Staubli VAL3: Cognex.pjx

--- Cognex.pjx ---
Parameters version=s7.4 stackSize=5000 millimeterUnit=true
Program file=checkCellFormat.pgx
Program file=checkColValue.pgx
Program file=checkErrFormat.pgx
Program file=debugMsg.pgx
Program file=example.pgx
Program file=getErrorCode.pgx
Program file=getErrorMessage.pgx
Program file=getFile.pgx
Program file=getFullError.pgx
Program file=getLibVersion.pgx
Program file=getNextID.pgx
Program file=getOnline.pgx
Program file=incrementCol.pgx
Program file=init.pgx
Program file=initPUPITRE.pgx
Program file=isIDAvailable.pgx
Program file=isLoggedIn.pgx
Program file=loadFile.pgx
Program file=login.pgx
Program file=programmeMOVE.pgx
Program file=readLogin.pgx
Program file=readNumValue.pgx
Program file=readRect.pgx
Program file=readSocket.pgx
Program file=readStrValue.pgx
Program file=readTrsf.pgx
Program file=readme.pgx
Program file=safety.pgx
Program file=saveFile.pgx
Program file=sendCommand.pgx
Program file=setCheckRow.pgx
Program file=setEventAndWait.pgx
Program file=setEventNoWait.pgx
Program file=setIDAutoMgt.pgx
Program file=setOnline.pgx
Program file=start.pgx
Program file=stop.pgx
Program file=trigger.pgx
Program file=writeFloatValue.pgx
Program file=writeIntValue.pgx
Program file=writeSocket.pgx
Program file=writeStrValue.pgx
Data file=Cognex.dtx
Type name=camera path=./camera/camera.pjx

--- checkCellFormat.pgx ---
public program checkCellFormat(num x_nCamID (dimensions=1), string& x_sCellNumber[] (dimensions=1), bool& x_bMatchOk[] (dimensions=1))
  local num l_i
  local bool l_bColOk
  local bool l_bRowOk
  local string l_sColumn
  local string l_sRow
  local num l_nRow
  local num l_nError
  local string l_sMsgError
begin
  //-----------------------------------------------------------------------
  //Header begin
  //Description of program
  // This routines checks if the format of the string used to point on a cell
  // of the cognex speadsheet matches the format of native command.
  //
  // Input Parameters
  //  x_nCamID :
  //    role : camera's ID
  //   x_sCellNumber  :
  //     role : Cell number in string format.
  //            Must be : - First digit is a letter (A-Z) for Column number
  //                      - 3 next digits is a number for Row number
  //
  // Output Parameteres
  //  x_bMatchOK  :
  //    role : retruns true if format of the string x_sCellNumber is correct
  //          and false otherwise.
  //
  //Examples
  //  call checkCellFormat(nCamID,"A3",l_bCellOk)
  //
  //Header end
  //-----------------------------------------------------------------------

  //Init
  x_bMatchOk=false
  //Verify length of the string (minimum 2 digit, ex : "A1")
  if len(x_sCellNumber)>=2
    //Column of the CellNumber
    l_sColumn=left(x_sCellNumber,1)
    //Verify first digit (column)
    //First digit must be in range 'A-Z' or 'a-z'
    call checkColValue(l_sColumn,l_bColOk)
    if l_bColOk
      //First digit OK
      //Row of the CellNumber
      l_sRow=right(x_sCellNumber,len(x_sCellNumber)-1)
      toNum(l_sRow,l_nRow,l_bRowOk)
      if l_bRowOk
        //l_sRow is a numercial value
        //Verify the row number
        if l_nRow>=0 and (l_nRow<=400 or !bCheckRowUpLim)
          if len(l_sRow)<3
            //Add digits (there is always 3 digits)
            l_sRow=left("000",3-len(l_sRow))+l_sRow
            //Update CellNumber
            x_sCellNumber=l_sColumn+l_sRow
          endIf
          //Cell Format OK
          x_bMatchOk=true
          cCamera[x_nCamID].nErrorCode=110
        else
          //Row number out of range
          cCamera[x_nCamID].nErrorCode=113
          cCamera[x_nCamID].sErrorMsg[cCamera[x_nCamID].nErrorCode]="Cell Format> "+l_sRow+" row number out of range"
        endIf
      else
        //Invalid row (not a numerical value)
        cCamera[x_nCamID].nErrorCode=112
        cCamera[x_nCamID].sErrorMsg[cCamera[x_nCamID].nErrorCode]="Cell Format> "+l_sRow+" invalid row"
      endIf
    else
      //Invalid column
      cCamera[x_nCamID].nErrorCode=111
      cCamera[x_nCamID].sErrorMsg[cCamera[x_nCamID].nErrorCode]="Cell Format> "+l_sColumn+" invalid column"
    endIf
  endIf
  if bDebugProgram
    //Displays error message
    call getFullError(x_nCamID,l_nError,l_sMsgError)
    ? l_sMsgError
  endIf
end

--- checkColValue.pgx ---
public program checkColValue(string x_sColCharac (dimensions=1), bool& x_bColOk[] (dimensions=1))
begin
  //-----------------------------------------------------------------------
  //Header begin
  //Description of program
  //  Check the column number of the x_sCellNumber.
  //
  // Input Parameters
  //   x_sCellNumber  :
  //     role : cell number in string format.
  //            Must be : - First digit is a letter (A-Z) for Column number
  //                      - 3 next digits is a number for Row number
  //
  // Output Parameteres
  //  x_bColOk  :
  //    role : returns true if the operation succeeded and false
  //          otherwise
  //
  //Header end
  //-----------------------------------------------------------------------

  //Verify column character (between "A" to "Z" or "a" to "z")
  x_bColOk=(asc(x_sColCharac,0)>=asc("a",0)) and (asc(x_sColCharac,0)<=asc("z",0))
  x_bColOk=x_bColOk or (asc(x_sColCharac,0)>=asc("A",0)) and (asc(x_sColCharac,0)<=asc("Z",0))
end

--- getErrorCode.pgx ---
public program getErrorCode(num x_nCamID (dimensions=1), num& x_nErrorCode[] (dimensions=1))
begin
  //-----------------------------------------------------------------------
  //Header begin
  //Description of program
  //  Get error code of last executed command.
  //
  //Input parameters
  //  num x_nCamID :
  //    role : camera's ID
  //
  //Output parameters
  //  num x_nErrorCode :
  //    role : error code of the last executed command
  //
  //Examples
  //  call getErrorCode(nCamID,l_nErrorCode)
  //
  //History
  //  Creation : 19-05-08 - f.Rob
  //  Modification 06-2012 - T.Caille - C.Rocchini
  //Header end
  //-----------------------------------------------------------------------
  if nLibErrorCode==0
    x_nErrorCode=cCamera[x_nCamID].nErrorCode
  else
    x_nErrorCode=nLibErrorCode
    nLibErrorCode=0
  endIf
  nCamID=x_nCamID
end

--- getLibVersion.pgx ---
public program getLibVersion(string& x_sVersion[] (dimensions=1))
begin
  //-----------------------------------------------------------------------
  //Header begin
  //Description of program
  //  Retrieve version of the library.
  //
  //Output parameters
  //  string x_sVersion :
  //    role : version of the library
  //
  //Examples
  //  call getLibVersion(l_sLibVersion)
  //
  //History
  //  Creation : 19-05-08 - f.Rob
  //Header end
  //-----------------------------------------------------------------------

  x_sVersion=strVersion
end

--- incrementCol.pgx ---
public program incrementCol(string& x_sCellNumber[] (dimensions=1), bool& x_bColumnOK[] (dimensions=1))
  local string l_sColCharac
begin
  //-----------------------------------------------------------------------
  //Header begin
  //Description of program
  //  Increment the column number of the x_sCellNumber.
  //
  // Input Parameters
  //   x_sCellNumber  :
  //     role : Cell number in string format.
  //            Must be : - First digit is a letter (A-Z) for Column number
  //                      - 3 next digits is a number for Row number
  //
  // Output Parameteres
  //  x_bColumnOK  :
  //    role : returns true if the increment column is succeeded and false
  //          otherwise
  //
  //History
  //  Creation : 19-05-08 - f.Rob
  //  Modification : 10-07-08 - CROC
  //    correction of bug in the line that rebuilds the new incremented cell
  //    number, the line "right(x_sCellNumber,3)" has been replaced by
  //    "right(x_sCellNumber,len(x_sCellNumber)-1)" to be more flexible in
  //    regards to cell number format (before that the cell number had to be
  //    composed of one letter and 3 numbers, now the only restriction is that
  //    the first character has to be a letter). This modification was triggered
  //    by the fact that this procedure is used by readRect() that passes the
  //    cell numbers as 2 char only (one letter, one number), thus it wasn't
  //    working properly.
  //Header end
  //-----------------------------------------------------------------------

  //Get the number column
  l_sColCharac=left(x_sCellNumber,1)
  //Increment the number column
  l_sColCharac=chr((asc(l_sColCharac,0)+1))
  //Checks the number column ( A<Column<Z)
  call checkColValue(l_sColCharac,x_bColumnOK)
  if x_bColumnOK
    //Modify x_sCellNumber
    x_sCellNumber=l_sColCharac+right(x_sCellNumber,len(x_sCellNumber)-1)
  endIf
end

--- loadFile.pgx ---
public program loadFile(num x_nCamID (dimensions=1), string x_sNameJob (dimensions=1), bool& x_bError[] (dimensions=1))
begin
  //-----------------------------------------------------------------------
  //Header begin
  //Description of program
  //  Loads the specified job from flash memory on the In-Sight sensor,
  //  making it the active job.
  //
  //!!! The In-Sight sensor must be OFFLINE !!!
  //
  //Input parameters
  //  num x_nCamID :
  //    role : camera's ID
  //
  //Output parameters
  //  string x_sNameJob :
  //    role : The name of the job.
  //           The command will execute with or without the .JOB extension.
  //
  //  bool x_bError :
  //    role : returns true if an error occurred and false otherwise
  //
  //Examples
  //   call loadFile(nCamID,"Camera1.job",x_bError)
  //
  //History
  //  Creation : 19-05-08 - f.Rob
  //Header end
  //-----------------------------------------------------------------------

  nProgram[x_nCamID]=4
  call sendCommand(x_nCamID,"LF"+x_sNameJob,x_bError)
end

--- login.pgx ---
public program login(sio& x_sioSocket (dimensions=1), string x_sUser (dimensions=1), string x_sPassword (dimensions=1), num& x_nCamID (dimensions=1), bool& x_bError[] (dimensions=1))
  local string l_sMsg
  local bool l_bError
begin
  //-----------------------------------------------------------------------
  //Header begin
  //Description of program
  //  Login to camera via TCP/IP socket port 1023, password pair
  // (usually "admin" and "").
  //  Returns camera's ID of type num for further communication with the camera.
  //
  //Input parameters
  //  string x_sUser :
  //    role : user name
  //  string x_sPassword :
  //    role : password for the user x_sUser
  //
  //Output parameters
  //  sio x_sioSocket :
  //    role : CS8 client socket
  //  num x_nCamID :
  //    role : returns camera's ID for further operations as the lib can
  //          communicate with more that 1 camera.
  //    posssible values : - first camera (first login)  : x_nCamID=1
  //                       - second camera (second login): x_nCamID=2
  //                       - ...
  //  bool x_bError :
  //    role : returns true if an error occurred and false otherwise
  //
  //Examples
  //  call login(cognex1,"admin","",nCamID,x_bError)
  //
  //History
  //  Creation : 19-05-08 - f.Rob
  //Header end
  //-----------------------------------------------------------------------
  if bDebugProgram
    putln("Cognex login")
  endIf
  // Check available ID
  l_bError=false
  if bGetID==true
    call isIDAvailable(x_nCamID,l_bError)
  endIf
  if l_bError==false
    nProgram[x_nCamID]=1
    sioLink(cCamera[x_nCamID].sSocket,x_sioSocket)
    // Read welcome string
    call readSocket(x_nCamID,l_sMsg,x_bError)
    // Send user name
    call readLogin(x_nCamID,l_sMsg,x_bError)
    call writeSocket(x_nCamID,x_sUser)
    // Send password
    call readLogin(x_nCamID,l_sMsg,x_bError)
    call writeSocket(x_nCamID,x_sPassword)
    // Read login result
    call readSocket(x_nCamID,l_sMsg,x_bError)
    x_bError=find(l_sMsg,"User Logged In")==-1
    if x_bError
      cCamera[x_nCamID].nErrorCode=1
      cCamera[x_nCamID].bConnected=false
      if bDebugProgram
        putln("Login : failed")
      endIf
    else
      cCamera[x_nCamID].bConnected=true
    endIf
  else
    x_bError=true
    nLibErrorCode=203
  endIf
end

--- programmeMOVE.pgx ---
program programmeMOVE()
begin
  while true

    // boucle infini

    while (borange==true)
      // BOUCLE DE DEBOXAGE

      // DEMANDE UNE MISE EN LIGNE DE LA CAMERA SI CELLE SI EST ETEINTE
      call getOnline(nCamID,resultTrigger)
      //APPEL UNE CAPURE DE PHOTO
      call trigger(nCamID,l_bError)

      delay(1.5)



      // RECUPERATION DONNE DANS LE TABLEUR COGNEX DANS LES CELLULE CC36/D36/E36
      call readNumValue(nCamID,"C36",resultx,l_bError)
      call readNumValue(nCamID,"D36",resulty,l_bError)
      call readNumValue(nCamID,"E36",resultz,l_bError)


      nbPoint=nbPoint+1
      putln("COORDONNEE DU POINT :")
      putln(nbPoint)
      putln("Coordonnée X:")
      putln(resultx)
      putln("Coordonnée Y:")
      putln(resulty)
      putln("Coordonnée Z:")
      putln(resultz)


      // AFFECTATION DES VALEUR DE X Y Z DU POINT CAMERA QUI EST DANS LE FRAME CAMERA
      PointCamera.trsf.x=resultx
      PointCamera.trsf.y=resulty
      PointCamera.trsf.z=55.5
      PointCamera.trsf.rx=180
      PointCamera.trsf.ry=0
      PointCamera.trsf.rz=90



      close(pince)



      movej(appro(PointCamera,{0,0,-100,0,0,0}),pince,rapide)
      movel(PointCamera,pince,lent)




      delay(1)

      open(pince)

      delay(1)


      movel(appro(PointCamera,{0,0,-100,0,0,0}),pince,rapide)
      movej(PointDePassage,pince,rapide)


      movej(PointDePoseHaut,pince,rapide)


      // attendre de fin de mouvement avant l'instruction suivante
      vvert=true

      //voyant vert passe a vrai
      wait(bvert!=false)

      // attend que bouton vert passe a vrai
      vvert=false
      movel(PointDePose,pince,lent)

      delay(1)
      close(pince)
      delay(1)

      movel(PointDePoseHaut,pince,lent)
      waitEndMove()


    endWhile
    call initPUPITRE()
    // appel le programme Init pour changement de rack.

  endWhile
end

--- readLogin.pgx ---
program readLogin(num x_nCamID (dimensions=1), string& x_sMsg[] (dimensions=1), bool& x_bError[] (dimensions=1))
  local num l_nChar
  local num l_nCount
begin
  //-----------------------------------------------------------------------
  //Header begin
  //Description of program
  // Read characters from socket until ":" is received
  //
  //Input parameters
  //  num x_nCamID :
  //    role : camera's ID
  //
  //Output parameters
  //  string x_sMsg:
  //    role : returns the error message
  //  bool x_bError :
  //    role : returns true if an error occurred and false otherwise
  //
  //Examples
  //  call readLogin(nCamID,"D5",l_nValue,x_bError)
  //
  //History
  //  Creation : 19-05-08 - f.Rob
  //Header end
  //-----------------------------------------------------------------------

  x_sMsg=""
  do
    l_nCount=sioGet(cCamera[x_nCamID].sSocket,l_nChar)
    //-1 : timeout for input communication has been reached
    if (l_nCount>-1) and (l_nChar>=32)
      x_sMsg=x_sMsg+chr(l_nChar)
    endIf
    x_bError=l_nCount<=-1
  until (chr(l_nChar)==":") or x_bError
  //Communication Error
  if x_bError
    cCamera[x_nCamID].nErrorCode=2
  endIf
  //Displays error message
  if bDebugProgram
    putln("ReadLogin : "+x_sMsg)
  endIf
end

--- readNumValue.pgx ---
public program readNumValue(num x_nCamID (dimensions=1), string x_sCellNumber (dimensions=1), num& x_nValue[] (dimensions=1), bool& x_bError[] (dimensions=1))
  local bool l_bIsOk
  local string l_sValue
  local string l_sMsgError
begin
  //-----------------------------------------------------------------------
  //Header begin
  //Description of program
  //  Read contents of a cell adressed by x_sCellNumber from camera's ID
  //  and convert it in numerical value.
  //
  //Input parameters
  //  num x_nCamID :
  //    role : camera's ID
  //  string x_sCellNumber :
  //    role : The column letter and the row number of the cell value to get.
  //    possible values : - column letter : (A to Z)
  //                      - row number : (000 to 399)
  //
  //Output parameters
  //  num x_nValue :
  //    role : contents of cell convert in numerical
  //  bool x_bError :
  //    role : returns true if an error occurred and false otherwise
  //
  //Examples
  //  call readNumValue(nCamID,"D5",l_nValue,x_bError)
  //
  //History
  //  Creation : 19-05-08 - f.Rob
  //  Modification : 10-07-08 - CROC
  //    inversion of returned error boolean, it was backwards (x_bError was
  //    set as the third param of the toNum(...) which is set to true when
  //    the toNum(...) worked OK, however x_bError needed to be true when
  //    the toNum(...) did not work OK.
  //Header end
  //-----------------------------------------------------------------------

  // Read contents of cell and transform it to a numerical value
  call readStrValue(x_nCamID,x_sCellNumber,l_sValue,x_bError)
  if !x_bError
    toNum(l_sValue,x_nValue,l_bIsOk)
    x_bError=!l_bIsOk
  endIf
end

--- setCheckRow.pgx ---
public program setCheckRow(bool x_bCheckUpLim (dimensions=1))
begin
  //-----------------------------------------------------------------------
  //Header begin
  //Description of program
  // This routines activates of de-activates the row number checking parameter
  // This parameter determines wether or not the row number will be checked against
  // the upper limit (400). The check against the lower limit (0) always remains active.
  //
  // Input Parameters
  //  x_bCheckUpLim :
  //    role : set to true to check row number against upper limit of 400 or to false otherwise
  //
  //Examples
  //  call setCheckRow(true)
  //
  //History
  //  Creation : 03-05-11 - CROC
  //Header end
  //-----------------------------------------------------------------------
  bCheckRowUpLim=x_bCheckUpLim
end

--- setIDAutoMgt.pgx ---
public program setIDAutoMgt(bool x_bAutoOn (dimensions=1))
begin
  //-----------------------------------------------------------------------
  //Header begin
  //Description of program
  //  Turn on/off automatic ID managment
  //  This routine should be called once when starting main application.
  //
  //Input parameters
  //  bool x_bAutoOn : enable/disable automatic ID managment
  //
  //Examples
  //  call setIDAutoMgt(true)
  //
  //History
  //  Creation : 12-12 - CROC
  //Header end
  //-----------------------------------------------------------------------
  bGetID=x_bAutoOn
end

--- trigger.pgx ---
public program trigger(num x_nCamID (dimensions=1), bool& x_bError[] (dimensions=1))
begin
  //-----------------------------------------------------------------------
  //Header begin
  //Description of program
  // Acquire a new image and evaluate it on the camera.
  //
  //Input parameters
  //  num x_nCamID :
  //    role : camera's ID
  //
  //Output parameters
  //  bool x_bError :
  //    role : returns true if an error occurred and false otherwise
  //
  //Examples
  //  call trigger(nCamID,l_bError)
  //
  //History
  //  Creation : 19-05-08 - f.Rob
  //Header end
  //-----------------------------------------------------------------------

  //Trigger image acquire and evaluation
  call setEventAndWait(x_nCamID,8,x_bError)
end

--- writeFloatValue.pgx ---
public program writeFloatValue(num x_nCamID (dimensions=1), string x_sCellNumber (dimensions=1), num x_nValue (dimensions=1), bool& x_bError[] (dimensions=1))
  local string l_sCell
  local bool l_bIsOk
begin
  //-----------------------------------------------------------------------
  //Header begin
  //Description of program
  //  Sets an edit box control contained in a cell (x_sCellNumber)
  //  to a specified floating-point value (x_nValue)
  //  The target cell of the writing operation in the Cognex spreadsheet must
  //  be of the EditFloat type.
  //
  //Input parameters
  //  num x_nCamID :
  //    role : camera's ID
  //  string x_sCellNumber :
  //    role : The column letter and the row number of the cell value to get.
  //    possible values : - column letter : (A to Z)
  //                      - row number : (000 to 399)
  //  num x_nValue :
  //    role : value to writing in the cell
  //
  //Output parameters
  //  bool x_bError :
  //    role : returns true if an error occurred and false otherwise
  //
  //Examples
  //  call writeFloatValue(nCamID,"C6",5.6,l_bError)
  //
  //History
  //  Creation : 19-05-08 - f.Rob
  //Header end
  //-----------------------------------------------------------------------

  // Write a float value into a cell
  x_bError=true
  call checkCellFormat(x_nCamID,x_sCellNumber,l_bIsOk)
  if l_bIsOk
    nProgram[x_nCamID]=9
    call sendCommand(x_nCamID,"SF"+x_sCellNumber+toString("0.5",x_nValue),x_bError)
  endIf
end

--- writeSocket.pgx ---
program writeSocket(num x_nCamID (dimensions=1), string x_sMsg (dimensions=1))
  local num i
begin
  //-----------------------------------------------------------------------
  //Header begin
  //Description of program
  //  Write string to socket character by character.
  //
  //Input parameters
  //  num x_nCamID :
  //    role : camera's ID
  //  string x_sMsg :
  //    role : native command
  //
  //Examples
  //  call sendCommand(nCamID,sCmd)
  //
  //History
  //  Creation : 19-05-08 - f.Rob
  //Header end
  //-----------------------------------------------------------------------

  for i=0 to (len(x_sMsg)-1)
    sioSet(cCamera[x_nCamID].sSocket,asc(x_sMsg,i))
  endFor
  sioSet(cCamera[x_nCamID].sSocket,13)
  sioSet(cCamera[x_nCamID].sSocket,10)
  if bDebugSocket
    ? "W Status code: "+x_sMsg
  endIf
end

--- writeStrValue.pgx ---
public program writeStrValue(num x_nCamID (dimensions=1), string x_sCellNumber (dimensions=1), string x_sMsg (dimensions=1), bool& x_bError[] (dimensions=1))
  local string l_sCell
  local bool l_bIsOk
begin
  //-----------------------------------------------------------------------
  //Header begin
  //Description of program
  //  Sets an edit box control contained in a cell (x_sCellNumber) to a
  //  specified string (x_sMsg)
  //  The target cell of the writing operation in the Cognex spreadsheet must
  //  be of the EditString type.
  //
  //Input parameters
  //  num x_nCamID :
  //    role : camera's ID
  //  string x_sCellNumber :
  //    role : The column letter and the row number of the cell value to get.
  //    possible values : - column letter : (A to Z)
  //                      - row number : (000 to 399)
  //  string x_sMsg :
  //    role : string to writing in the cell
  //
  //Output parameters
  //  bool x_bError :
  //    role : returns false if operation suceeded and true otherwise
  //
  //Examples
  //  call writeStrValue(nCamID,"C6","Example Staubli",l_bError)
  //
  //History
  //  Creation : 19-05-08 - f.Rob
  //Header end
  //-----------------------------------------------------------------------

  x_bError=true
  call checkCellFormat(x_nCamID,x_sCellNumber,l_bIsOk)
  if l_bIsOk
    nProgram[x_nCamID]=11
    call sendCommand(x_nCamID,"SS"+x_sCellNumber+x_sMsg,x_bError)
  endIf
end
